TYPE DataBuffer :
STRUCT
	WIDP : DINT;
	PmcData : DUT_St0Data;
	stPLCData 			: DUT_stPLCData;
END_STRUCT
END_TYPE

(* stored: Version 1.1.0.1, ProductVersion 3.1.4024.15
   DUT DataBuffer: Id {bfcac84a-b92e-4729-99c7-020ef0d05817} *)
